// LS Electric XG5000 project: MOV
// PLC LSPLC
// module base 0 slot 0: 입출력 모듈:XBC-DR30S (DC 24V 입력 18점, 릴레이 출력 12점)

PROGRAM MOV (task: 스캔 프로그램)

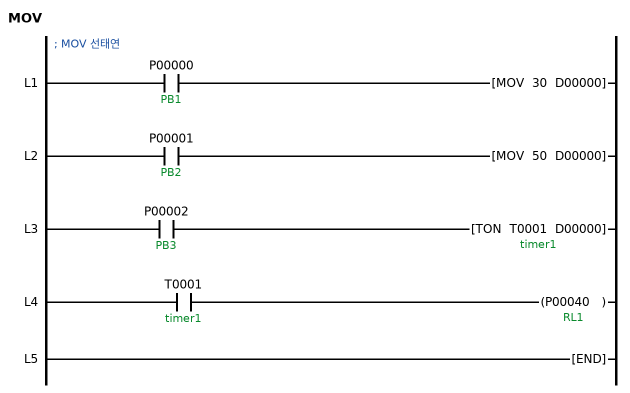
// MOV 선태연
; L1
LOAD      P00000	// PB1
MOV       30 D00000
; L2
LOAD      P00001	// PB2
MOV       50 D00000
; L3
LOAD      P00002	// PB3
TON       T0001 D00000	// timer1
; L4
LOAD      T0001	// timer1
OUT       P00040	// RL1
; L5
END